FUNCTION_BLOCK FB_Object
VAR_INPUT
END_VAR
VAR_OUTPUT
END_VAR
VAR
END_VAR

PROPERTY Index : int
GET
END_GET
SET
END_SET
END_PROPERTY

PROPERTY IsEnabled : bool
GET
END_GET
SET
END_SET
END_PROPERTY

END_FUNCTION_BLOCK

(* stored: Version 1.1.0.1, ProductVersion 3.1.4024.11
   POU FB_Object: Id {b5cde4e1-0d3d-4cec-9ffd-a4b8d7366ca7}, SpecialFunc None
   Property Index: Id {3dee1e96-bba9-4682-8032-9c9b591f0f26}
   Get Get: Id {51f1c38d-d294-4e08-a558-cd9f7e9dd460}
   Set Set: Id {ee8fc1b6-417e-4f91-a117-e6c246cdadeb}
   Property IsEnabled: Id {2a44d89f-58c4-47bd-924f-d35123939f43}
   Get Get: Id {9daf83a8-ab2a-46ac-a755-167f27f5a86e}
   Set Set: Id {861925f1-fcb3-404f-b975-f6abd1d94937} *)
